(* IEC 61131-3 sources: RL_MAR/experiments/comparison/llm4plc/results/gpt-4o_20260507_114630/20260507_121216, 1 file *)

(* ---- generated_code_iteration_0.st ---- *)
```pascal
START_ST
FUNCTION_BLOCK TheaterControl
VAR_INPUT
    StartButton : BOOL; (* Input for starting a performance *)
    StopButton : BOOL; (* Input for stopping a performance *)
    SceneNumber : INT; (* Input for selecting the scene or act *)
END_VAR
VAR_OUTPUT
    LightingControl : BOOL; (* Output for controlling lighting *)
    SoundControl : BOOL; (* Output for controlling sound *)
    PerformanceInProgress : BOOL; (* Indicator for an ongoing performance *)
END_VAR
VAR
    state : INT; (* Current state of the system *)
    prevState : INT; (* Previous state of the system *)
END_VAR

(* Initialize outputs and states *)
IF NOT (StartButton OR StopButton) THEN
    IF state = 0 THEN
        (* STATE 0: IDLE *)
        LightingControl := FALSE;
        SoundControl := FALSE;
        PerformanceInProgress := FALSE;
        IF StartButton THEN
            state := 1;
        END_IF;
ENDIF
END_ST
